Universal Robots PolyScope program: g01_pp_cycle_only.urp

Program g01_pp_cycle_only (installation=default directory=/programs createdIn=5.9.1.1031110 lastSavedIn=5.9.1.1031110 robotSerialNumber=20195501059)
Calibrated DH parameters: a=[0.000146, -0.418764, -0.053981, 0.000058, -0.000023, 0]; d=[0.162545, 37.319448, -206.067439, 168.881546, 0.09955, 0.099464]; alpha=[1.57004, -0.001979, 0.002304, 1.570607, -1.57066, 0]; deltaTheta=[0, -0.174616, -1.258233, 1.432844, -0.000001, 0]
BeforeStart
  URCap Gripper Activate (Robotiq_Grippers, Robotiq Inc.) dataModel(ResetAndActivateKey=false)
Robot Program (runOnlyOnce=false)
  URCap Grip Check (Robotiq_Grippers, Robotiq Inc.) dataModel(ObjectDetectedKey=true, DimensionValidationKey=false, DimensionKey=100.0, DimensionDimensionPositiveGapKey=5.0, DimensionNegativeGapKey=5.0, GripperIdKey=1, ModelDefinedKey=true); state(isChildrenLocked=true)
    URCap If (Robotiq_Grippers, Robotiq Inc.)
      Call g01_nut_dropoff
    URCap Else (Robotiq_Grippers, Robotiq Inc.)
      Call g01_nut_pickup_1
      Call g01_home_1
SubProgram  [hidden by the author, left out]
SubProgram -> g01_nut_pickup_1
SubProgram  [hidden by the author, left out]
SubProgram g01_nut_dropoff [hidden by the author, left out]
SubProgram g01_nut_pickup_1 (keepSynchronizedWithDisk=true) programFile=/programs/g01_nut_pickup.urp
  URCap Grip Check (Robotiq_Grippers, Robotiq Inc.) dataModel(DimensionDimensionPositiveGapKey=5.0, DimensionNegativeGapKey=5.0, GripperIdKey=1, ModelDefinedKey=true, ObjectDetectedKey=true, DimensionKey=75.76078431372548, DimensionValidationKey=false); state(isChildrenLocked=true)
    URCap If (Robotiq_Grippers, Robotiq Inc.)
      Halt
  URCap Gripper (Robotiq_Grippers, Robotiq Inc.) dataModel(position=100.0, force=100.0, speed=100.0, positionInDouble=100.0, forceInDouble=100.0, speedInDouble=100.0, slaveIds=[9], blocking=true)
  MoveL speed 250 mm/s, acceleration 1200 mm/s^2 (useActiveTCP=true) feature=Base
    Waypoint Waypoint (Variable): variable(featureName=g01_nut_pickup)
    MoveDirectionNode (selectedDirection=ZPlus toolParams=0.02, 1.2) feature=Joint_6_name
      Until DISTANCE (allowActions=true deceleration=3 distanceNodeType=STOP) Distance=0.01; motionParameters(blendRadius=0)
        Waypoint Waypoint (Variable): variable(featureName=g01_nut_pickup)
        Popup Error (haltProgram=false message=No nut inputType=Text)
      Until TOOL_CONTACT_DETECTION (allowActions=true retraction=0.002 decelerationAcceleration=1 decelerationAngularAcceleration=34.906585)
        URCap Gripper (Robotiq_Grippers, Robotiq Inc.) dataModel(position=59.29411764705882, force=100.0, speed=100.0, positionInDouble=59.29411764705882, forceInDouble=100.0, speedInDouble=100.0, slaveIds=[9], blocking=true)
        MoveDirectionNode (selectedDirection=ZPlus toolParams=0.02, 1.2) feature=Joint_6_name
          Until TOOL_CONTACT_DETECTION (allowActions=false retraction=0 decelerationAcceleration=3 decelerationAngularAcceleration=34.906585)
        URCap Gripper (Robotiq_Grippers, Robotiq Inc.) dataModel(position=100.0, force=100.0, speed=100.0, positionInDouble=100.0, forceInDouble=100.0, speedInDouble=100.0, slaveIds=[9], blocking=true)
        URCap Gripper (Robotiq_Grippers, Robotiq Inc.) dataModel(position=64.76575362969615, force=100.0, speed=100.0, positionInDouble=64.76575362969615, forceInDouble=100.0, speedInDouble=100.0, slaveIds=[9], blocking=true)
        Script file /programs/rot90.script
          | q = get_joint_positions()
          | # move 1/4 of a turn...
          | q[5] = q[5] + d2r(90)
          | movej(q)
        URCap Gripper (Robotiq_Grippers, Robotiq Inc.) dataModel(position=100.0, force=100.0, speed=100.0, positionInDouble=100.0, forceInDouble=100.0, speedInDouble=100.0, slaveIds=[9], blocking=true)
        URCap Gripper (Robotiq_Grippers, Robotiq Inc.) dataModel(position=64.76575362969615, force=100.0, speed=100.0, positionInDouble=64.76575362969615, forceInDouble=100.0, speedInDouble=100.0, slaveIds=[9], blocking=true)
        Script file /programs/nut_pick_trick.script
          | q = get_joint_positions()
          | # move 1/24 of a turn... try not to grip on peaks
          | q[5] = q[5] + d2r(360/24)
          | movej(q)
        URCap Gripper (Robotiq_Grippers, Robotiq Inc.) dataModel(position=100.0, force=100.0, speed=100.0, positionInDouble=100.0, forceInDouble=100.0, speedInDouble=100.0, slaveIds=[9], blocking=true)
    Waypoint Waypoint (Variable): variable(featureName=g01_nut_pickup)
SubProgram g01_home_1 [hidden by the author, left out]
